// TIA Portal V17 export
Cycle "Codex_Cycle_3s"  CycleTime=3, CycleUnit=Second, StartingPoint=****-**-**T**:**:**, Comment="Codex cycle import/export loop test."
